FUNCTION_BLOCK FB_HwRefInterlockBase
VAR_INPUT
END_VAR
VAR_OUTPUT
	eCurrentState : E_InterlockState := E_InterlockState.Locked;
END_VAR
VAR
END_VAR

METHOD M_LockUnlock : ERRORID
VAR_INPUT
	bLock : BOOL;
END_VAR
IF bLock THEN
	eCurrentState := E_InterlockState.Locked;
ELSE
	eCurrentState := E_InterlockState.Unlocked;
END_IF
END_METHOD

END_FUNCTION_BLOCK

(* stored: Version 1.1.0.1, ProductVersion 3.1.4022.7
   POU FB_HwRefInterlockBase: Id {b5db477d-5c7e-44a0-92a7-31f4293dad49}, SpecialFunc None
   Method M_LockUnlock: Id {397d4a1e-5405-4a50-bdc3-32af3a942589} *)
